(* PLC project PLCOpen_Leer.project, CODESYS CODESYS V3.5 SP7 Patch 2 *)
(* stored: creationDateTime 2018-07-08T13:58:46.9898301, modificationDateTime 2018-07-08T13:57:47.963454 *)

VAR_GLOBAL  (* globalVarList *)
  Step_1 : BOOL;
  deactStep_1 : BOOL;
  actStep_1 : BOOL;
  Step_3 : BOOL;
  deactStep_3 : BOOL;
  actStep_3 : BOOL;
  deactEnStep_4 : BOOL;
  EnStep_4 : BOOL;
  actEnStep_4 : BOOL;
  Step_5 : BOOL;
  deactStep_5 : BOOL;
  actStep_5 : BOOL;
  Step_2 : BOOL;
  deactStep_2 : BOOL;
  actStep_2 : BOOL;
END_VAR

PROGRAM GlobalFB
  VAR_INPUT
    End : BOOL;
    Init : BOOL;
    Enable : BOOL;
  END_VAR
  VAR
    TransLoop : INT;
    NumTrans : INT;
    stableState : BOOL;
    T_2 : BOOL;
    T_1 : BOOL;
    T_3 : BOOL;
    T_4 : BOOL;
  END_VAR

		  	  
		  		IF enable THEN
		  			WHILE  DO
		  			IF (NOT(init))AND(NOT(end)) THEN
		  				IF (DI_2)AND(T_2) THEN
		  					stableState := true;
		  					actStep_3 := true;
		  					Step_3 := true;
		  					deactStep_3 := false;
		  					actStep_2 := false;
		  					deactStep_2 := true;
		  					Step_2 := false;
		  				END_IF
		  				IF ((actStep_1)AND(Step_1)AND(deactStep_1)) THEN
		  					IF actStep_1 THEN
		  						actStep_1 := false;
		  					END_IF
		  					IF deactStep_1 THEN
		  						deactStep_1 := false;
		  					END_IF
		  					IF Step_1 THEN
		  						;
		  					END_IF
		  				END_IF
		  				IF ((actStep_3)AND(Step_3)AND(deactStep_3)) THEN
		  					IF actStep_3 THEN
		  						actStep_3 := false;
		  					END_IF
		  					IF deactStep_3 THEN
		  						deactStep_3 := false;
		  					END_IF
		  					IF Step_3 THEN
		  						;
		  					END_IF
		  				END_IF
		  				IF ((actEnStep_4)AND(EnStep_4)AND(deactEnStep_4)) THEN
		  					IF deactEnStep_4 THEN
		  						deactEnStep_4 := false;
		  					END_IF
		  					IF actEnStep_4 THEN
		  						actEnStep_4 := false;
		  					END_IF
		  					IF EnStep_4 THEN
		  						;
		  					END_IF
		  				END_IF
		  				IF ((actStep_5)AND(Step_5)AND(deactStep_5)) THEN
		  					IF actStep_5 THEN
		  						actStep_5 := false;
		  					END_IF
		  					IF deactStep_5 THEN
		  						deactStep_5 := false;
		  					END_IF
		  					IF Step_5 THEN
		  						;
		  					END_IF
		  				END_IF
		  				IF (DI_1)AND(T_1) THEN
		  					stableState := true;
		  					actStep_1 := false;
		  					deactStep_1 := true;
		  					Step_1 := false;
		  					EnStep_4 := true;
		  					actEnStep_4 := true;
		  					deactEnStep_4 := false;
		  					deactStep_2 := false;
		  					Step_2 := true;
		  					actStep_2 := true;
		  				END_IF
		  				T_1 := Step_1;
		  				IF (DI_3)AND(T_3) THEN
		  					stableState := true;
		  					actStep_5 := true;
		  					Step_5 := true;
		  					deactStep_5 := false;
		  					actEnStep_4 := false;
		  					deactEnStep_4 := true;
		  					EnStep_4 := false;
		  					Step_3 := false;
		  					deactStep_3 := true;
		  					actStep_3 := false;
		  				END_IF
		  				IF (true)AND(T_4) THEN
		  					stableState := true;
		  					actStep_5 := false;
		  					deactStep_5 := true;
		  					Step_5 := false;
		  					actStep_1 := true;
		  					Step_1 := true;
		  					deactStep_1 := false;
		  				END_IF
		  				T_3 := (TRUE);
		  				IF ((actStep_2)AND(Step_2)AND(deactStep_2)) THEN
		  					IF actStep_2 THEN
		  						actStep_2 := false;
		  					END_IF
		  					IF deactStep_2 THEN
		  						deactStep_2 := false;
		  					END_IF
		  					IF Step_2 THEN
		  						;
		  					END_IF
		  				END_IF
		  				T_4 := Step_5;
		  				T_2 := Step_2;
		  			END_IF
		  			TransLoop := (TransLoop+1);
		  			stableState := false;
		  			END_WHILE;
		  			TransLoop := (0);
		  		END_IF
		  		IF init THEN
		  			Step_1 := false;
		  			actStep_1 := false;
		  			deactStep_1 := false;
		  			actStep_3 := false;
		  			deactStep_3 := false;
		  			Step_3 := false;
		  			EnStep_4 := true;
		  			deactEnStep_4 := false;
		  			actEnStep_4 := false;
		  			actStep_5 := false;
		  			deactStep_5 := false;
		  			Step_5 := false;
		  			actStep_2 := false;
		  			deactStep_2 := false;
		  			Step_2 := false;
		  		END_IF
		  		IF end THEN
		  			actStep_1 := false;
		  			deactStep_1 := false;
		  			Step_1 := false;
		  			Step_3 := false;
		  			actStep_3 := false;
		  			deactStep_3 := false;
		  			deactEnStep_4 := false;
		  			actEnStep_4 := false;
		  			EnStep_4 := false;
		  			Step_5 := false;
		  			actStep_5 := false;
		  			deactStep_5 := false;
		  			Step_2 := false;
		  			actStep_2 := false;
		  			deactStep_2 := false;
		  		END_IF
		  		
		  	  
		  	
END_PROGRAM
